SUBAPPLICATION Softkey_IXA_TO_Remote_WRITE_BG_OPC (* VT-SoftKey lesen (ODER lokaler Web-Override, z.B. vt-ui-mirror auf demselben Modul) + Remote-OPC-UA-Write an Zielmodul + VT-Hintergrundfarbe aus Remote-Subscribe (generisch, ein Kanal, fuer Funktionen ohne lokalen physischen Ausgang - Bedienung sitzt auf STG1, Aktor auf einem Modul ohne eigene VT-Anbindung) *)
  (* Standard: 61499-2 *)
  (* Version 1.0, 2026-09-05, franz, Meisterschulen am Ostbahnhof *)
  PACKAGE MyLib::sys;
  IMPORT isobus::UT::Q::const::IDs::ID_NULL;
  (* Documentation:
  SoftKey → Remote-OPC-UA-Write mit Status-Feedback (ein Kanal)
   Für Funktionen, deren Bedienung auf einem VT-Steuergerät (STG1) sitzt, deren Aktor aber auf einem anderen Modul ohne eigene VT-Anbindung liegt: der lokale SoftKey löst per OPC-UA einen Remote-Write zum Zielmodul aus, und der tatsächliche Zustand kommt per Remote-Subscribe zurück und wird als Hintergrundfarbe direkt am SoftKey angezeigt.
   Funktionsbeschreibung
    - Softkey_IXA liest den lokalen SoftKey (u16ObjId).
   - SUBSCRIBE_WEB (ID_WEB_READ) erlaubt zusätzlich einem lokalen Web-Client (z.B. vt-ui-mirror auf demselben Modul) dieselbe Funktion auszulösen - OR_MERGE (AX_OR_2) verknüpft SoftKey und Web-Override per ODER.
   - AX_CLIENT_1_0 (ID_WRITE_REMOTE) schreibt das gemergte Signal per OPC-UA an das Zielmodul.
   - AX_SUBSCRIBE_1 (ID_SUBSCRIBE) empfängt den tatsächlichen Zustand vom Zielmodul zurück und speist ihn in GreenWhiteBackground1_AX - ein normales VT-Objekt genügt hier ein Q_BackgroundColour-Kommando.
    Kommt am Zielobjekt auch ein Auxiliary-Function-Objekt (Joystick) ins Spiel, Softkey_Aux_IXA_TO_Remote_WRITE_BG_OPC verwenden (dieselbe Struktur, zusätzlich eine dritte Quelle und GreenWhiteBackground3_AX statt 1_AX). Für einen VT-Button statt SoftKey Button_IXA_TO_Remote_WRITE_BG_OPC.
  *)
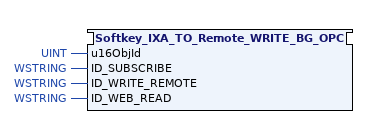
  VAR_INPUT
    u16ObjId : UINT := ID_NULL; (* Object ID SoftKey/Hintergrund (VT) *)
    ID_SUBSCRIBE : WSTRING; (* Remote-Subscribe-Adresse (Status/Farbe, ACTION=SUBSCRIBE) *)
    ID_WRITE_REMOTE : WSTRING; (* Remote-Write-Adresse zum Zielmodul (Befehl, ACTION=WRITE, CLIENT) *)
    ID_WEB_READ : WSTRING; (* Lokale Subscribe-Adresse fuer einen Web-Client (z.B. vt-ui-mirror) auf demselben Modul, ODER-verknuepft mit dem echten SoftKey *)
  END_VAR
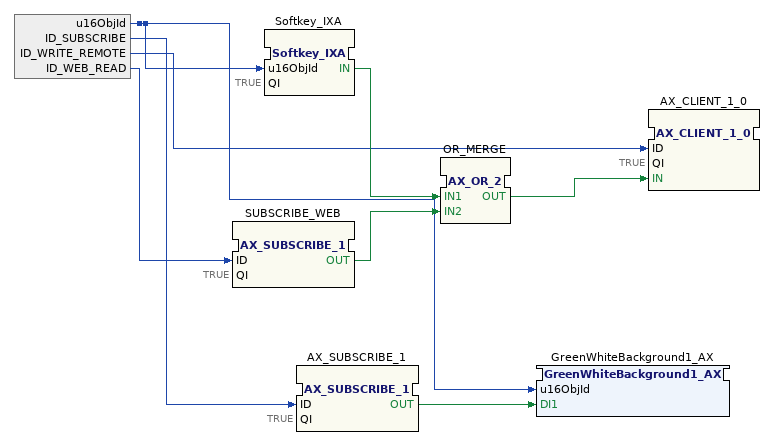
  FBS
    Softkey_IXA : isobus::UT::io::Softkey::Softkey_IXA(QI := TRUE);
    SUBSCRIBE_WEB : adapter::net::AX_SUBSCRIBE_1(QI := TRUE);
    OR_MERGE : adapter::booleanOperators::AX_OR_2;
    AX_CLIENT_1_0 : adapter::net::AX_CLIENT_1_0(QI := TRUE);
    AX_SUBSCRIBE_1 : adapter::net::AX_SUBSCRIBE_1(QI := TRUE);
  END_FBS
  SUBAPPS
    GreenWhiteBackground1_AX : MyLib::sys::GreenWhiteBackground1_AX;
  END_SUBAPPS
  DATA_CONNECTIONS
    u16ObjId TO Softkey_IXA.u16ObjId;
    u16ObjId TO GreenWhiteBackground1_AX.u16ObjId;
    ID_WEB_READ TO SUBSCRIBE_WEB.ID;
    ID_SUBSCRIBE TO AX_SUBSCRIBE_1.ID;
    ID_WRITE_REMOTE TO AX_CLIENT_1_0.ID;
  END_CONNECTIONS
  ADAPTER_CONNECTIONS
    Softkey_IXA.IN TO OR_MERGE.IN1;
    SUBSCRIBE_WEB.OUT TO OR_MERGE.IN2;
    OR_MERGE.OUT TO AX_CLIENT_1_0.IN;
    AX_SUBSCRIBE_1.OUT TO GreenWhiteBackground1_AX.DI1;
  END_CONNECTIONS
END_SUBAPPLICATION
